FUNCTION_BLOCK ABSTRACT AbstractState IMPLEMENTS I_State
VAR_INPUT
	ipStatehandler: I_Statehandler;
END_VAR
VAR
	fbTON: TON;
END_VAR

METHOD FB_init : BOOL
VAR_INPUT
	bInitRetains : BOOL; // if TRUE, the retain variables are initialized (warm start / cold start)
	bInCopyCode : BOOL;  // if TRUE, the instance afterwards gets moved into the copy code (online change)
	ipStatehandler: I_Statehandler;
END_VAR
THIS^.ipStatehandler := ipStatehandler;
END_METHOD

METHOD ABSTRACT Handle : BOOL
END_METHOD

END_FUNCTION_BLOCK

(* stored: Version 1.1.0.1, ProductVersion 3.1.4024.3
   POU AbstractState: Id {fa262302-fbab-4380-bea0-f5c030f48e7a}, SpecialFunc None
   Method FB_init: Id {e82d3211-c556-47a7-a96b-fd256a0d2ee5}
   Method Handle: Id {74617af7-e3cd-4159-9f51-aa4c332d44e9} *)
